{attribute 'qualified_only'}
VAR_GLOBAL CONSTANT
	
(*
			============================GENERAL SHUTTER LAYOUT===============================
			  ________________________________________________________________________________
	        ||                                  HALL SWITCH                                   \
	X- side ||       ----14---13--12---11---10---9---8---7---6---5---4---3---2--1---0----      \    X+ side
			||_________________________________________________________________________         \	
			| | 				 |                 **  **  **                 |        \ MotorXP \
			| |					 |            *                  *            |         \ MotorXM \   
			| |					 |         *                        *         |          \_________\
			| |				     |       *                            *       |                   | |
			| |					 |      *                              *      |                   | |
			| |		     	     |     *                                *     |                   | |
			| |		BLADE 	     |     *            APERTURE            *     |       BLADE       | |
			| |		STACK	     |     *                                *     |       STACK       | |
			| |		 XM 	     |     *                                *     |        XP         | |
			| |					 |      *                              *      |                   | |
			| |					 |       *                            *       |                   | |
			| |					 |         *                        *         |                   | |
			| |					 |   	      *                  *            |                   | |
			|_|__________________|_________________**  **  **_________________|___________________|_|
			
			       ---Negative-Direction--->                          <---Positive-Direction---
*)

	 
	cHallLower 		: INT := 0;
	cHallUpper 		: INT := 14;
	cDirPos			: INT := 0;
	cDirNeg			: INT := 1;
	cTripPerHall	: INT := 16;
	cNumOfHall		: INT := 15;
	cTripCount		: INT := (cTripPerHall*cNumOfHall)-1;
	cMio0           : INT := 0;  // Identifies the first multi-timestamping digital I/O module, MIO-00.
	cMio1           : INT := 1;  // Identifies the second MIO module, MIO-01.
	cFirstMio1Hall  : INT := 8;  // Hall sensors with this ID or greater are on the second MIO, MIO-01.
	  
	cBrakeOff		: BOOL	:= TRUE;
	cBrakeOn		: BOOL	:= FALSE;
	cScanVel		: LREAL := 30;//60;
	cHomeVel		: LREAL	:= 1;
	cCalibrateVel	: LREAL	:= 100;
	cPositionVel	: LREAL := 300;
	cPosStart		: LREAL := 0;
	cPosEnd			: LREAL := 750.76; //this will need to change for production once keyance snesors are in
	
	//For indexing axis
	cXP : INT := 0;  // +X side.
	cXM : INT := 1;  // -X side.
	
	// For how many cycles should we save PLC external task-start time and MIO SysTimes?
	cTimeBufferDepth: INT := 5;
	
	// Version number for the set of messages passsing between CCS and this firmware.
	nVersion		: DINT := 3;
	
END_VAR
VAR_GLOBAL
	//Safety State
	bSafetyOn	: BOOL := TRUE;
	
	//Hall Switches
	nHallSequence 			: WORD;
		
	// We're using our MIOs in synchronous multi-timestamping mode with a Multi-TimeStamping Factor (MTSF) of 2x. We expect at most one Hall event
	// per channel per cycle, so we've set the MTSF to 2x as recommended by the EL12xx manual.
	
	// SysTime is a 64-bit variable that in multi-timestamp mode contains the lower 32 bits of the MIO's DC clock. Each MIO channel reacts to a state change
	// by generating a timestamp that's a copy of the lower 32 bits of the current SysTime.
	
	{attribute 'TcLinkTo' := '[0] := TIID^Device 1 (EtherCAT)^MCD-00 (EK1200)^MIO-00 (EL1259)^DEV Inputs Device^SysTime;
	                          [1] := TIID^Device 1 (EtherCAT)^MCD-00 (EK1200)^MIO-01 (EL1259)^DEV Inputs Device^SysTime'}
	mioSysTime AT %I*: ARRAY [GVL.cMio0 .. GVL.cMio1] OF ULINT;  

	// The first event timestamp for each MIO channel that we use.
	{attribute 'TcLinkTo' := '
     [0]  := TIID^Device 1 (EtherCAT)^MCD-00 (EK1200)^MIO-00 (EL1259)^MTI Inputs 2x Channel 1^Input event time 1;
	 [1]  := TIID^Device 1 (EtherCAT)^MCD-00 (EK1200)^MIO-00 (EL1259)^MTI Inputs 2x Channel 2^Input event time 1;
	 [2]  := TIID^Device 1 (EtherCAT)^MCD-00 (EK1200)^MIO-00 (EL1259)^MTI Inputs 2x Channel 3^Input event time 1;
	 [3]  := TIID^Device 1 (EtherCAT)^MCD-00 (EK1200)^MIO-00 (EL1259)^MTI Inputs 2x Channel 4^Input event time 1;
	 [4]  := TIID^Device 1 (EtherCAT)^MCD-00 (EK1200)^MIO-00 (EL1259)^MTI Inputs 2x Channel 5^Input event time 1;
	 [5]  := TIID^Device 1 (EtherCAT)^MCD-00 (EK1200)^MIO-00 (EL1259)^MTI Inputs 2x Channel 6^Input event time 1;
	 [6]  := TIID^Device 1 (EtherCAT)^MCD-00 (EK1200)^MIO-00 (EL1259)^MTI Inputs 2x Channel 7^Input event time 1;
	 [7]  := TIID^Device 1 (EtherCAT)^MCD-00 (EK1200)^MIO-00 (EL1259)^MTI Inputs 2x Channel 8^Input event time 1;
	 [8]  := TIID^Device 1 (EtherCAT)^MCD-00 (EK1200)^MIO-01 (EL1259)^MTI Inputs 2x Channel 1^Input event time 1;
	 [9]  := TIID^Device 1 (EtherCAT)^MCD-00 (EK1200)^MIO-01 (EL1259)^MTI Inputs 2x Channel 2^Input event time 1;
	 [10] := TIID^Device 1 (EtherCAT)^MCD-00 (EK1200)^MIO-01 (EL1259)^MTI Inputs 2x Channel 3^Input event time 1;
	 [11] := TIID^Device 1 (EtherCAT)^MCD-00 (EK1200)^MIO-01 (EL1259)^MTI Inputs 2x Channel 4^Input event time 1;
	 [12] := TIID^Device 1 (EtherCAT)^MCD-00 (EK1200)^MIO-01 (EL1259)^MTI Inputs 2x Channel 5^Input event time 1;
	 [13] := TIID^Device 1 (EtherCAT)^MCD-00 (EK1200)^MIO-01 (EL1259)^MTI Inputs 2x Channel 6^Input event time 1;
	 [14] := TIID^Device 1 (EtherCAT)^MCD-00 (EK1200)^MIO-01 (EL1259)^MTI Inputs 2x Channel 7^Input event time 1'}
	nInputEventTime	AT %I*	: ARRAY [cHallLower .. cHallUpper] OF UDINT;

	// The input event count for each MIO channel that we use.
	{attribute 'TcLinkTo' := '
     [0]  := TIID^Device 1 (EtherCAT)^MCD-00 (EK1200)^MIO-00 (EL1259)^MTI Inputs 2x Channel 1^No of input events;
	 [1]  := TIID^Device 1 (EtherCAT)^MCD-00 (EK1200)^MIO-00 (EL1259)^MTI Inputs 2x Channel 2^No of input events;
	 [2]  := TIID^Device 1 (EtherCAT)^MCD-00 (EK1200)^MIO-00 (EL1259)^MTI Inputs 2x Channel 3^No of input events;
	 [3]  := TIID^Device 1 (EtherCAT)^MCD-00 (EK1200)^MIO-00 (EL1259)^MTI Inputs 2x Channel 4^No of input events;
	 [4]  := TIID^Device 1 (EtherCAT)^MCD-00 (EK1200)^MIO-00 (EL1259)^MTI Inputs 2x Channel 5^No of input events;
	 [5]  := TIID^Device 1 (EtherCAT)^MCD-00 (EK1200)^MIO-00 (EL1259)^MTI Inputs 2x Channel 6^No of input events;
	 [6]  := TIID^Device 1 (EtherCAT)^MCD-00 (EK1200)^MIO-00 (EL1259)^MTI Inputs 2x Channel 7^No of input events;
	 [7]  := TIID^Device 1 (EtherCAT)^MCD-00 (EK1200)^MIO-00 (EL1259)^MTI Inputs 2x Channel 8^No of input events;
	 [8]  := TIID^Device 1 (EtherCAT)^MCD-00 (EK1200)^MIO-01 (EL1259)^MTI Inputs 2x Channel 1^No of input events;
	 [9]  := TIID^Device 1 (EtherCAT)^MCD-00 (EK1200)^MIO-01 (EL1259)^MTI Inputs 2x Channel 2^No of input events;
	 [10] := TIID^Device 1 (EtherCAT)^MCD-00 (EK1200)^MIO-01 (EL1259)^MTI Inputs 2x Channel 3^No of input events;
	 [11] := TIID^Device 1 (EtherCAT)^MCD-00 (EK1200)^MIO-01 (EL1259)^MTI Inputs 2x Channel 4^No of input events;
	 [12] := TIID^Device 1 (EtherCAT)^MCD-00 (EK1200)^MIO-01 (EL1259)^MTI Inputs 2x Channel 5^No of input events;
	 [13] := TIID^Device 1 (EtherCAT)^MCD-00 (EK1200)^MIO-01 (EL1259)^MTI Inputs 2x Channel 6^No of input events;
	 [14] := TIID^Device 1 (EtherCAT)^MCD-00 (EK1200)^MIO-01 (EL1259)^MTI Inputs 2x Channel 7^No of input events'}
	nNumOfInputs AT %I*		: ARRAY [cHallLower .. cHallUpper] OF USINT;

	// Indicates for each channel whether the event was caused by a rising (1) or a falling (0) edge.
	{attribute 'TcLinkTo' := '
    [0]  := TIID^Device 1 (EtherCAT)^MCD-00 (EK1200)^MIO-00 (EL1259)^MTI Inputs 2x Channel 1^Input event state 1;
	[1]  := TIID^Device 1 (EtherCAT)^MCD-00 (EK1200)^MIO-00 (EL1259)^MTI Inputs 2x Channel 2^Input event state 1;
	[2]  := TIID^Device 1 (EtherCAT)^MCD-00 (EK1200)^MIO-00 (EL1259)^MTI Inputs 2x Channel 3^Input event state 1;
	[3]  := TIID^Device 1 (EtherCAT)^MCD-00 (EK1200)^MIO-00 (EL1259)^MTI Inputs 2x Channel 4^Input event state 1;
	[4]  := TIID^Device 1 (EtherCAT)^MCD-00 (EK1200)^MIO-00 (EL1259)^MTI Inputs 2x Channel 5^Input event state 1;
	[5]  := TIID^Device 1 (EtherCAT)^MCD-00 (EK1200)^MIO-00 (EL1259)^MTI Inputs 2x Channel 6^Input event state 1;
	[6]  := TIID^Device 1 (EtherCAT)^MCD-00 (EK1200)^MIO-00 (EL1259)^MTI Inputs 2x Channel 7^Input event state 1;
	[7]  := TIID^Device 1 (EtherCAT)^MCD-00 (EK1200)^MIO-00 (EL1259)^MTI Inputs 2x Channel 8^Input event state 1;
	[8]  := TIID^Device 1 (EtherCAT)^MCD-00 (EK1200)^MIO-01 (EL1259)^MTI Inputs 2x Channel 1^Input event state 1;
	[9]  := TIID^Device 1 (EtherCAT)^MCD-00 (EK1200)^MIO-01 (EL1259)^MTI Inputs 2x Channel 2^Input event state 1;
	[10] := TIID^Device 1 (EtherCAT)^MCD-00 (EK1200)^MIO-01 (EL1259)^MTI Inputs 2x Channel 3^Input event state 1;
	[11] := TIID^Device 1 (EtherCAT)^MCD-00 (EK1200)^MIO-01 (EL1259)^MTI Inputs 2x Channel 4^Input event state 1;
	[12] := TIID^Device 1 (EtherCAT)^MCD-00 (EK1200)^MIO-01 (EL1259)^MTI Inputs 2x Channel 5^Input event state 1;
	[13] := TIID^Device 1 (EtherCAT)^MCD-00 (EK1200)^MIO-01 (EL1259)^MTI Inputs 2x Channel 6^Input event state 1;
	[14] := TIID^Device 1 (EtherCAT)^MCD-00 (EK1200)^MIO-01 (EL1259)^MTI Inputs 2x Channel 7^Input event state 1'}
	bInputEventState AT %I*	: ARRAY [cHallLower .. cHallUpper] OF BOOL;

	//Timer
	fbWaitTimer	: TON;
	
	//TestVariable
	fbWritePersistentData	: WritePersistentData;
	
	// Process data from the EtherCAT master. The time offset types are given as ULINT instead of LINT because
	// that's how the corresponding arguments to F_GetCurExtTime64() are declared.
	{attribute 'TcLinkTo' :=  'TIID^Device 1 (EtherCAT)^InfoData^DcToExtTimeOffset'}
	DcToExtTimeOffset AT %I*: ULINT;

    {attribute 'TcLinkTo' :=  'TIID^Device 1 (EtherCAT)^InfoData^DcToTcTimeOffset'}
	DcToTcTimeOffset AT %I*: ULINT;
	
	// Process data from the EL6688 PTP module, MTM-00.
	{attribute 'TcLinkTo' := 'TIID^Device 1 (EtherCAT)^MCD-00 (EK1200)^MTM-00 (EL6688)^InfoData^AdsAddr'}
	ptpAdsAddr AT %I*: AMSADDR;       // Used to contact the module for CoE data.


END_VAR

VAR_GLOBAL PERSISTENT // For million cycle test
	strokeXP	: UDINT;
	strokeXM	: UDINT;
END_VAR

(* stored: Version 1.1.0.1, ProductVersion 3.1.4022.18
   GVL GVL: Id {543590d2-21dc-426c-bb1c-cff8b9e02654} *)
